// TIA Portal project "IMPERIAL" (V15)
// CUBE 67+ && PLC SIEMENS && ROBOT && PANTALLA GP-PRO

(* hardware
DEVICE "ROBOT1"  SIMATIC PC station
   slot 0: "Estación PC"  Rail  SIMATIC PC-Station  V1.0
      slot 125: "Stationmanager"  Station_Manager  V6.0.4
   slot 1: "CP 1616_1"  CP 1616  6GK1 161-6AA00  V2.6
DEVICE "Dispositivo GSD_1"  GSD.Device.PN
   slot 0: "Rack"  Rack  V1.0
   slot 0: "Cube67-BN-PNIO"  Cube67+ BN-PNIO  56526  2
      slot 0: "Cube67+ BN-PNIO_1"  Cube67+ BN-PNIO
      slot 1: "Cube67+ BN-PNIO"  Cube67+ BN-PNIO
         slot 1: "Puerto 1"  Port 1
         slot 2: "Puerto 2"  Port 2
      slot 1: "Alimentación de energía_1"  Power Supply
         slot 0: "Alimentación de energía"  Power Supply
   slot 3: "Rama 1_1"  Branch 0
      slot 0: "Rama 1"  Branch 0
   slot 4: "56601 DIO16 E 8xM12_1"  56601 DIO16 E 8xM12  56601
      slot 0: "56601 DIO16 E 8xM12"  56601 DIO16 E 8xM12
   slot 5: "Rama 2_1"  Branch 1
      slot 0: "Rama 2"  Branch 1
   slot 6: "56600 DIO16 C 8xM12_1"  56600 DIO16 C 8xM12  56600
      slot 0: "56600 DIO16 C 8xM12"  56600 DIO16 C 8xM12
   slot 7: "Rama 3_1"  Branch 2
      slot 0: "Rama 3"  Branch 2
   slot 8: "Rama 4_1"  Branch 3
      slot 0: "Rama 4"  Branch 3
DEVICE "S7-1200 station_1"  S7-1200 Station
   slot 0: "Rack_0"  S7-1200 Rack  Rack  V1.0
   slot 1: "PLC_1"  CPU 1212C DC/DC/DC  6ES7 212-1AE40-0XB0  V4.2
*)

// ===== PLC "PLC_1"  CPU 1212C DC/DC/DC =====

VAR_GLOBAL   // PLC tag table "Tabla de variables estándar"
   "PLC_C67_FOT_DAR_DARSENA2" AT %I29.7 : Bool;   // FOTO ESPEJO DAR 2
   "PLC_67_SME_DAR_DARSENA1" AT %I23.7 : Bool;   // FOTO DARSENA 1
   "R01_PLC_ORD_EXT_MDZ" AT %I10.0 : Bool;
   "R01_PLC_ORD_RET_MDZ" AT %I10.1 : Bool;
   "R01_PLC_PROD_COG_T1" AT %I10.2 : Bool;
   "NºSACOS" AT %IW30 : Word;
   "Nº DEJADAS CAPA PAR" AT %IW32 : Word;
   "Nº DEJADA CAPA IMPAR" AT %IW34 : Word;
   "ANCHO SACO" AT %IW36 : Word;
   "LARGO SACO" AT %IW38 : Word;
   "ALTO SACO" AT %IW40 : Word;
   "ANCHO PALET" AT %IW42 : Word;
   "LARGO PALET" AT %IW44 : Word;
   "ALTO PALET" AT %IW46 : Word;
   "X" AT %IW48 : Word;
   "Y" AT %IW50 : Word;
   "GIRO" AT %IB51 : Byte;
   "COGIDA" AT %I52.0 : Bool;
   "X(1)" AT %IW130 : Word;
   "Y(1)" AT %IW132 : Word;
   "GIRO(1)" AT %IB134 : Byte;
   "COGIDA(1)" AT %I135.0 : Bool;
   "X(2)" AT %IW136 : Word;
   "Y(2)" AT %IW138 : Word;
   "GIRO(2)" AT %IB140 : Byte;
   "COGIDA(2)" AT %I141.0 : Bool;
   "X(3)" AT %IW142 : Word;
   "Y(3)" AT %IW144 : Word;
   "GIRO(3)" AT %IB146 : Byte;
   "COGIDA(3)" AT %I147.0 : Bool;
   "X(4)" AT %IW148 : Word;
   "Y(4)" AT %IW150 : Word;
   "GIRO(4)" AT %IB152 : Byte;
   "COGIDA(4)" AT %I153.0 : Bool;
   "X(5)" AT %IW154 : Word;
   "Y(5)" AT %IW156 : Word;
   "GIRO(5)" AT %IB158 : Byte;
   "COGIDA(5)" AT %I159.0 : Bool;
   "X(6)" AT %IW160 : Word;
   "Y(6)" AT %IW162 : Word;
   "GIRO(6)" AT %IB164 : Byte;
   "COGIDA(6)" AT %I165.0 : Bool;
   "X(7)" AT %IW166 : Word;
   "Y(7)" AT %IW168 : Word;
   "GIRO(7)" AT %IB170 : Byte;
   "COGIDA(7)" AT %I171.0 : Bool;
   "X(10)" AT %IW172 : Word;
   "Y(10)" AT %IW174 : Word;
   "GIRO(10)" AT %IB176 : Byte;
   "COGIDA(10)" AT %I177.0 : Bool;
   "X(11)" AT %IW178 : Word;
   "Y(11)" AT %IW180 : Word;
   "GIRO(11)" AT %IB182 : Byte;
   "COGIDA(11)" AT %I183.0 : Bool;
   "X(12)" AT %IW184 : Word;
   "Y(12)" AT %IW186 : Word;
   "GIRO(12)" AT %IB188 : Byte;
   "COGIDA(12)" AT %I189.0 : Bool;
   "X(13)" AT %IW190 : Word;
   "Y(13)" AT %IW192 : Word;
   "GIRO(13)" AT %IB194 : Byte;
   "COGIDA(13)" AT %I195.0 : Bool;
   "X(14)" AT %IW196 : Word;
   "Y(14)" AT %IW198 : Word;
   "GIRO(14)" AT %IB200 : Byte;
   "COGIDA(14)" AT %I201.0 : Bool;
   "X(15)" AT %IW202 : Word;
   "Y(15)" AT %IW204 : Word;
   "GIRO(15)" AT %IB206 : Byte;
   "COGIDA(15)" AT %I207.0 : Bool;
   "X(16)" AT %IW208 : Word;
   "Y(16)" AT %IW210 : Word;
   "GIRO(16)" AT %IB212 : Byte;
   "COGIDA(16)" AT %I213.0 : Bool;
   "X(17)" AT %IW214 : Word;
   "Y(17)" AT %IW216 : Word;
   "GIRO(17)" AT %IB218 : Byte;
   "COGIDA(17)" AT %I219.0 : Bool;
   "TE_TRANSPORT_1" AT %I220.0 : Bool;
   "TE_TRANSPORT_2" AT %I220.1 : Bool;
   "Programa_Activo" AT %I11.1 : Bool;
   "Seguridades_R01_OK" AT %I11.0 : Bool;
   "Botonera_Boton_Rojo" AT %I0.0 : Bool;
   "Botonera_Boton_Verde" AT %I0.1 : Bool;
   "Botonera_Boton_Amarillo" AT %I0.2 : Bool;
   "R01_PLC_PROD_COG_T2" AT %I10.3 : Bool;
   "R01_PLC_ORD_EXT_PIS" AT %I10.4 : Bool;
   "R01_PLC_ROB_COG_T1" AT %I10.5 : Bool;
   "R01_PLC_ROB_COG_T2" AT %I10.6 : Bool;
   "R01_PLC_ORDEN_ABRIR" AT %Q19.1 : Bool;
   "R01_PLC_ORDEN_CERRAR" AT %Q19.2 : Bool;
   "P_On" AT %Q29.3 : Bool;
   "RESET_FLANCO_SUB" AT %Q29.5 : Bool;
   "PLC_R01_PERM_COG_SACO_T1" AT %Q10.2 : Bool;
   "PLC_R01_PERM_COG_SACO_T2" AT %Q10.3 : Bool;
   "Botonera_Luz_Roja" AT %Q0.0 : Bool;
   "Botonera_Luz_Verde" AT %Q0.1 : Bool;
   "Botonera_Luz_Amarillo" AT %Q0.2 : Bool;
   "R01_Boton_Rojo" AT %Q12.0 : Bool;
   "R01_Boton_Verde" AT %Q12.1 : Bool;
   "R01_Boton_Amarilla" AT %Q12.2 : Bool;
   "PLC_R01_PIS_EXT" AT %Q10.4 : Bool;
   "Orden_Abrir_Mordaza" AT %M200.0 : Bool;
   "Orden_Cerrar_Mordaza" AT %M200.1 : Bool;
   "Tag_8" AT %M200.3 : Bool;
   "Tag_8(1)" AT %M201.4 : Bool;
   "Tag_9" AT %M201.6 : Bool;
   "Tag_12(1)" AT %M201.7 : Bool;
   "Tag_10" AT %M202.0 : Bool;
   "Tag_13" AT %M202.1 : Bool;
   "Tag_11" AT %M202.2 : Bool;
   "Tag_100" AT %M202.3 : Bool;
   "LUZ_AMARILLA" AT %M202.4 : Bool;
   "LUZ_ROJA" AT %M202.5 : Bool;
   "LUZ_VERDE" AT %M202.6 : Bool;
   "Permiso_Meter_Saco" AT %M202.7 : Bool;
   "ERROR_GLOBAL" AT %M203.0 : Bool;
   "Seguridades_Armadas" AT %M201.0 : Bool;
   "PLC_C67_MDZ_RET_GAR" AT %Q21.6 : Bool;
   "PLC_C67_MDZ_EXT_GAR" AT %Q21.4 : Bool;
   "PLC_C67_EXT_P1" AT %Q21.2 : Bool;
   "PLC_C67_EXT_P2" AT %Q21.0 : Bool;
   "C67_PLC_SME_P2_RET" AT %I20.3 : Bool;
   "C67_PLC_SME_P2_EXT" AT %I21.3 : Bool;
   "C67_PLC_SME_P1_RET" AT %I20.1 : Bool;
   "C67_PLC_SME_P1_EXT" AT %I21.1 : Bool;
   "C67_PLC_SME_GARR_RET" AT %I21.5 : Bool;
   "C67_PLC_SME_GARR_EXT" AT %I20.5 : Bool;
   "PLC_C67_EXT_COST" AT %Q22.2 : Bool;
   "PLC_C67_MOT1_AVAN" AT %Q22.0 : Bool;
   "PLC_C67_MOT1_RET" AT %Q23.0 : Bool;
   "C67_PLC_FOTO_INICIO" AT %I23.3 : Bool;
   "C67_PLC_FOTO_FIN" AT %I23.1 : Bool;
   "C67_PLC_SME_COST_EXT" AT %I23.5 : Bool;
   "C67_PLC_SME_COST_RET" AT %I22.5 : Bool;
   "Tag_1" AT %I11.5 : Bool;
   "Tag_2" AT %Q11.4 : Bool;
   "Tag_3" AT %Q11.2 : Bool;
   "PLC_R01_MDZ_EXT" AT %Q10.0 : Bool;
   "PLC_R01_MDZ_RET" AT %Q10.1 : Bool;
END_VAR

DATA_BLOCK "DB_1"   // DB1
{ S7_Optimized_Access := 'FALSE' }
VERSION : 0.1
   VAR
      GP_SysStartAddress : Int;
   END_VAR
BEGIN
END_DATA_BLOCK

DATA_BLOCK "PISTON_EV_DB_1"   // DB2
{ S7_Optimized_Access := 'TRUE' }
VERSION : 0.1
// stored: InstanceOfName PISTON_EV
"PISTON_EV"
BEGIN
END_DATA_BLOCK

DATA_BLOCK "FUNCION_COGER_R01_DB_1"   // DB3
{ S7_Optimized_Access := 'TRUE' }
VERSION : 0.1
// stored: InstanceOfName FUNCION_COGER_R01
"FUNCION_COGER_R01"
BEGIN
END_DATA_BLOCK

DATA_BLOCK "FUNCION_PISADOR_DB"   // DB4
{ S7_Optimized_Access := 'TRUE' }
VERSION : 0.1
// stored: InstanceOfName FUNCION_PISADOR
"FUNCION_PISADOR"
BEGIN
END_DATA_BLOCK

DATA_BLOCK "FUNCION_COGER_R01_DB"   // DB5
{ S7_Optimized_Access := 'TRUE' }
VERSION : 0.1
// stored: InstanceOfName FUNCION_COGER_R01
"FUNCION_COGER_R01"
BEGIN
END_DATA_BLOCK

DATA_BLOCK "FUNCION_EV_DB"   // DB6
{ S7_Optimized_Access := 'TRUE' }
VERSION : 0.1
// stored: InstanceOfName FUNCION_EV
"FUNCION_EV"
BEGIN
END_DATA_BLOCK

DATA_BLOCK "FUNCION_EV_DB_1"   // DB7
{ S7_Optimized_Access := 'TRUE' }
VERSION : 0.1
// stored: InstanceOfName FUNCION_EV
"FUNCION_EV"
BEGIN
END_DATA_BLOCK

DATA_BLOCK "FUNCION_PISADOR_DB_1"   // DB8
{ S7_Optimized_Access := 'TRUE' }
VERSION : 0.1
// stored: InstanceOfName FUNCION_PISADOR
"FUNCION_PISADOR"
BEGIN
END_DATA_BLOCK

DATA_BLOCK "FUNCION_PISADOR_1_DB"   // DB9
{ S7_Optimized_Access := 'TRUE' }
VERSION : 0.1
// stored: InstanceOfName FUNCION_PISADOR
"FUNCION_PISADOR"
BEGIN
END_DATA_BLOCK

DATA_BLOCK "FUNCION_PISADOR_2_DB"   // DB10
{ S7_Optimized_Access := 'TRUE' }
VERSION : 0.1
// stored: InstanceOfName FUNCION_PISADOR
"FUNCION_PISADOR"
BEGIN
END_DATA_BLOCK

DATA_BLOCK "PISTON_EV_DB_2"   // DB11
{ S7_Optimized_Access := 'TRUE' }
VERSION : 0.1
// stored: InstanceOfName PISTON_EV
"PISTON_EV"
BEGIN
END_DATA_BLOCK

DATA_BLOCK "PISTON_EV_DB_3"   // DB12
{ S7_Optimized_Access := 'TRUE' }
VERSION : 0.1
// stored: InstanceOfName PISTON_EV
"PISTON_EV"
BEGIN
END_DATA_BLOCK

DATA_BLOCK "FUNCION_COGER_R01_DB_2"   // DB13
{ S7_Optimized_Access := 'TRUE' }
VERSION : 0.1
// stored: InstanceOfName FUNCION_COGER_R01
"FUNCION_COGER_R01"
BEGIN
END_DATA_BLOCK

DATA_BLOCK "FUNCION_COGER_R01_DB_3"   // DB14
{ S7_Optimized_Access := 'TRUE' }
VERSION : 0.1
// stored: InstanceOfName FUNCION_COGER_R01
"FUNCION_COGER_R01"
BEGIN
END_DATA_BLOCK

DATA_BLOCK "FUNCION_COGER_R01_DB_4"   // DB15
{ S7_Optimized_Access := 'TRUE' }
VERSION : 0.1
// stored: InstanceOfName FUNCION_COGER_R01
"FUNCION_COGER_R01"
BEGIN
END_DATA_BLOCK

DATA_BLOCK "FUNCION_COGER_R01_DB_5"   // DB16
{ S7_Optimized_Access := 'TRUE' }
VERSION : 0.1
// stored: InstanceOfName FUNCION_COGER_R01
"FUNCION_COGER_R01"
BEGIN
END_DATA_BLOCK

DATA_BLOCK "FUNCION_EV_DB_2"   // DB17
{ S7_Optimized_Access := 'TRUE' }
VERSION : 0.1
// stored: InstanceOfName FUNCION_EV
"FUNCION_EV"
BEGIN
END_DATA_BLOCK

DATA_BLOCK "FUNCION_PISADOR_DB_2"   // DB18
{ S7_Optimized_Access := 'TRUE' }
VERSION : 0.1
// stored: InstanceOfName FUNCION_PISADOR
"FUNCION_PISADOR"
BEGIN
END_DATA_BLOCK

DATA_BLOCK "FUNCION_PISADOR_DB_3"   // DB19
{ S7_Optimized_Access := 'TRUE' }
VERSION : 0.1
// stored: InstanceOfName FUNCION_PISADOR
"FUNCION_PISADOR"
BEGIN
END_DATA_BLOCK

DATA_BLOCK "FUNCION_EV_DB_3"   // DB20
{ S7_Optimized_Access := 'TRUE' }
VERSION : 0.1
// stored: InstanceOfName FUNCION_EV
"FUNCION_EV"
BEGIN
END_DATA_BLOCK

DATA_BLOCK "FUNCION_COGER_R01_DB_6"   // DB21
{ S7_Optimized_Access := 'TRUE' }
VERSION : 0.1
// stored: InstanceOfName FUNCION_COGER_R01
"FUNCION_COGER_R01"
BEGIN
END_DATA_BLOCK

DATA_BLOCK "PISTON_EV_DB"   // DB23
{ S7_Optimized_Access := 'TRUE' }
VERSION : 0.1
// stored: InstanceOfName PISTON_EV
"PISTON_EV"
BEGIN
END_DATA_BLOCK

DATA_BLOCK "TRANSPORTADOR_AUTOMATICO_DB"   // DB24
{ S7_Optimized_Access := 'TRUE' }
VERSION : 0.1
// stored: InstanceOfName TRANSPORTADOR_AUTOMATICO
"TRANSPORTADOR_AUTOMATICO"
BEGIN
END_DATA_BLOCK

DATA_BLOCK "FUNCION_EV_DB_8"   // DB25
{ S7_Optimized_Access := 'TRUE' }
VERSION : 0.1
// stored: InstanceOfName FUNCION_EV
"FUNCION_EV"
BEGIN
END_DATA_BLOCK

DATA_BLOCK "FUNCION_EV_DB_9"   // DB26
{ S7_Optimized_Access := 'TRUE' }
VERSION : 0.1
// stored: InstanceOfName FUNCION_EV
"FUNCION_EV"
BEGIN
END_DATA_BLOCK

DATA_BLOCK "FUNCION_EV_DB_4"   // DB30
{ S7_Optimized_Access := 'TRUE' }
VERSION : 0.1
// stored: InstanceOfName FUNCION_EV
"FUNCION_EV"
BEGIN
END_DATA_BLOCK

DATA_BLOCK "FUNCION_EV_DB_5"   // DB31
{ S7_Optimized_Access := 'TRUE' }
VERSION : 0.1
// stored: InstanceOfName FUNCION_EV
"FUNCION_EV"
BEGIN
END_DATA_BLOCK

DATA_BLOCK "PISTON_EV_DB_4"   // DB32
{ S7_Optimized_Access := 'TRUE' }
VERSION : 0.1
// stored: InstanceOfName PISTON_EV
"PISTON_EV"
BEGIN
END_DATA_BLOCK

DATA_BLOCK "PISTON_EV_DB_5"   // DB33
{ S7_Optimized_Access := 'TRUE' }
VERSION : 0.1
// stored: InstanceOfName PISTON_EV
"PISTON_EV"
BEGIN
END_DATA_BLOCK

DATA_BLOCK "FUNCION_EV_DB_6"   // DB34
{ S7_Optimized_Access := 'TRUE' }
VERSION : 0.1
// stored: InstanceOfName FUNCION_EV
"FUNCION_EV"
BEGIN
END_DATA_BLOCK

DATA_BLOCK "FUNCION_EV_DB_7"   // DB35
{ S7_Optimized_Access := 'TRUE' }
VERSION : 0.1
// stored: InstanceOfName FUNCION_EV
"FUNCION_EV"
BEGIN
END_DATA_BLOCK

DATA_BLOCK "EMPUJADOR_DB"   // DB36
{ S7_Optimized_Access := 'TRUE' }
VERSION : 0.1
// stored: InstanceOfName EMPUJADOR
"EMPUJADOR"
BEGIN
END_DATA_BLOCK

DATA_BLOCK "TRANSPORTADOR_AUTOMATICO_DB_1"   // DB37
{ S7_Optimized_Access := 'TRUE' }
VERSION : 0.1
// stored: InstanceOfName TRANSPORTADOR_AUTOMATICO
"TRANSPORTADOR_AUTOMATICO"
BEGIN
END_DATA_BLOCK

DATA_BLOCK "TRANSPORTADOR_AUTOMATICO_DB_2"   // DB38
{ S7_Optimized_Access := 'TRUE' }
VERSION : 0.1
// stored: InstanceOfName TRANSPORTADOR_AUTOMATICO
"TRANSPORTADOR_AUTOMATICO"
BEGIN
END_DATA_BLOCK

DATA_BLOCK "TRANSPORTADOR_AUTOMATICO_DB_3"   // DB39
{ S7_Optimized_Access := 'TRUE' }
VERSION : 0.1
// stored: InstanceOfName TRANSPORTADOR_AUTOMATICO
"TRANSPORTADOR_AUTOMATICO"
BEGIN
END_DATA_BLOCK

DATA_BLOCK "TRANSPORTADOR_AUTOMATICO_DB_4"   // DB40
{ S7_Optimized_Access := 'TRUE' }
VERSION : 0.1
// stored: InstanceOfName TRANSPORTADOR_AUTOMATICO
"TRANSPORTADOR_AUTOMATICO"
BEGIN
END_DATA_BLOCK

DATA_BLOCK "TRANSPORTADOR_AUTOMATICO_DB_5"   // DB41
{ S7_Optimized_Access := 'TRUE' }
VERSION : 0.1
// stored: InstanceOfName TRANSPORTADOR_AUTOMATICO
"TRANSPORTADOR_AUTOMATICO"
BEGIN
END_DATA_BLOCK

DATA_BLOCK "TRANSPORTADOR_AUTOMATICO_DB_6"   // DB42
{ S7_Optimized_Access := 'TRUE' }
VERSION : 0.1
// stored: InstanceOfName TRANSPORTADOR_AUTOMATICO
"TRANSPORTADOR_AUTOMATICO"
BEGIN
END_DATA_BLOCK

FUNCTION_BLOCK "PISTON_EV"   // FB1, LAD
TITLE = EV
{ S7_Optimized_Access := 'TRUE' }
VERSION : 0.1
   VAR_INPUT
      ORDEN_EXTENDER : Bool;
      ORDEN_RETRAER : Bool;
      SENSOR_EXTENDIDO : Bool;
      SENSOR_RETRAIDO : Bool;
   END_VAR
   VAR_OUTPUT
      CILINDRO_EXTENDIDO : Bool;
      EXTENDER_CILINDRO : Bool;
      CILINDRO_RETRAIDO : Bool;
      RETRAER_CILINDRO : Bool;
   END_VAR
BEGIN

REGION Network 1
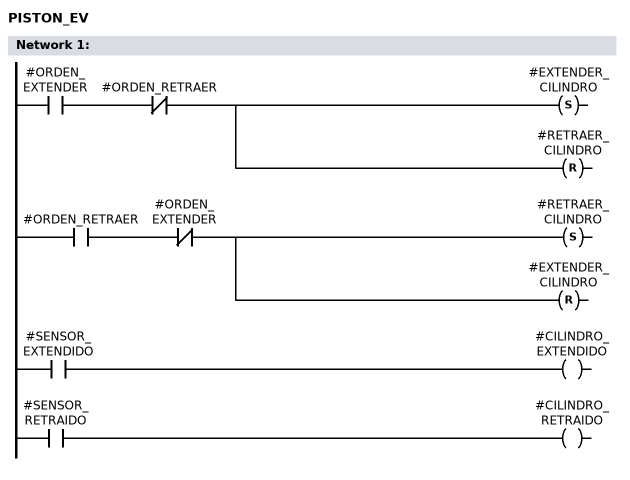
   RUNG wire#powerrail
      Contact( #ORDEN_EXTENDER )
      I_Contact( #ORDEN_RETRAER )
      wire#w1
      S_Coil( #EXTENDER_CILINDRO )
   END_RUNG
   RUNG wire#w1
      R_Coil( #RETRAER_CILINDRO )
   END_RUNG
   RUNG wire#powerrail
      Contact( #ORDEN_RETRAER )
      I_Contact( #ORDEN_EXTENDER )
      wire#w2
      S_Coil( #RETRAER_CILINDRO )
   END_RUNG
   RUNG wire#w2
      R_Coil( #EXTENDER_CILINDRO )
   END_RUNG
   RUNG wire#powerrail
      Contact( #SENSOR_EXTENDIDO )
      Coil( #CILINDRO_EXTENDIDO )
   END_RUNG
   RUNG wire#powerrail
      Contact( #SENSOR_RETRAIDO )
      Coil( #CILINDRO_RETRAIDO )
   END_RUNG
   // the same network as SCL:
   IF #ORDEN_EXTENDER AND NOT #ORDEN_RETRAER THEN
       #EXTENDER_CILINDRO := TRUE;
       #RETRAER_CILINDRO := FALSE;
   END_IF;
   IF #ORDEN_RETRAER AND NOT #ORDEN_EXTENDER THEN
       #RETRAER_CILINDRO := TRUE;
       #EXTENDER_CILINDRO := FALSE;
   END_IF;
   #CILINDRO_EXTENDIDO := #SENSOR_EXTENDIDO;
   #CILINDRO_RETRAIDO := #SENSOR_RETRAIDO;
END_REGION
END_FUNCTION_BLOCK

FUNCTION_BLOCK "FUNCION_EV"   // FB2, LAD
{ S7_Optimized_Access := 'TRUE' }
VERSION : 0.1
   VAR_INPUT
      Orden_Retraer_Pistones : Bool;   // INPUT
      Orden_Extender_Pistones : Bool;   // INPUT
      Sensor_1_Extendido : Bool;   // INPUT
      Sensor_1_Retraido : Bool;   // INPUT
      Sensor_2_Extendido : Bool;   // INPUT
      Sensor_2_Retraido : Bool;   // INPUT
      EN_Piston_Doble : Bool;   // INPUT
      EN_Switch_Final_Carrera_Retraer : Bool;   // INPUT
      EN_Switch_Final_Carrera_Extender : Bool;   // INPUT
      Tiempo_Error_Extender_100ms : Time := T#100ms;   // 0
      Tiempo_Error_Retraer_100ms : Time := T#100ms;   // 0
   END_VAR
   VAR_OUTPUT
      Error_Extender : Bool;   // OUTPUT
      Error_Retroceder : Bool;   // OUTPUT
      Extender_Pistones : Bool;
      Retraer_Pistones : Bool;
      Pistones_Retraidos : Bool;
      Pistones_Extendidos : Bool;
   END_VAR
   VAR
      Extender_Piston_1 : Bool;   // INTERNAL
      Extender_Piston_2 : Bool;   // INTERNAL
      Retraer_Piston_1 : Bool;   // INTERNAL
      Retraer_Piston_2 : Bool;   // INTERNAL
      Piston_1_Extendido : Bool;   // INTERNAL
      Piston_1_Retraido : Bool;   // INTERNAL
      Piston_2_Extendido : Bool;   // INTERNAL
      Piston_2_Retraido : Bool;   // INTERNAL
      Piston_1 : "PISTON_EV";
      Piston_2 : "PISTON_EV";
      Timer_1 : Time;   // INTERNAL
      Timer_2 : Time;   // INTERNAL
   END_VAR
BEGIN

REGION Network 1
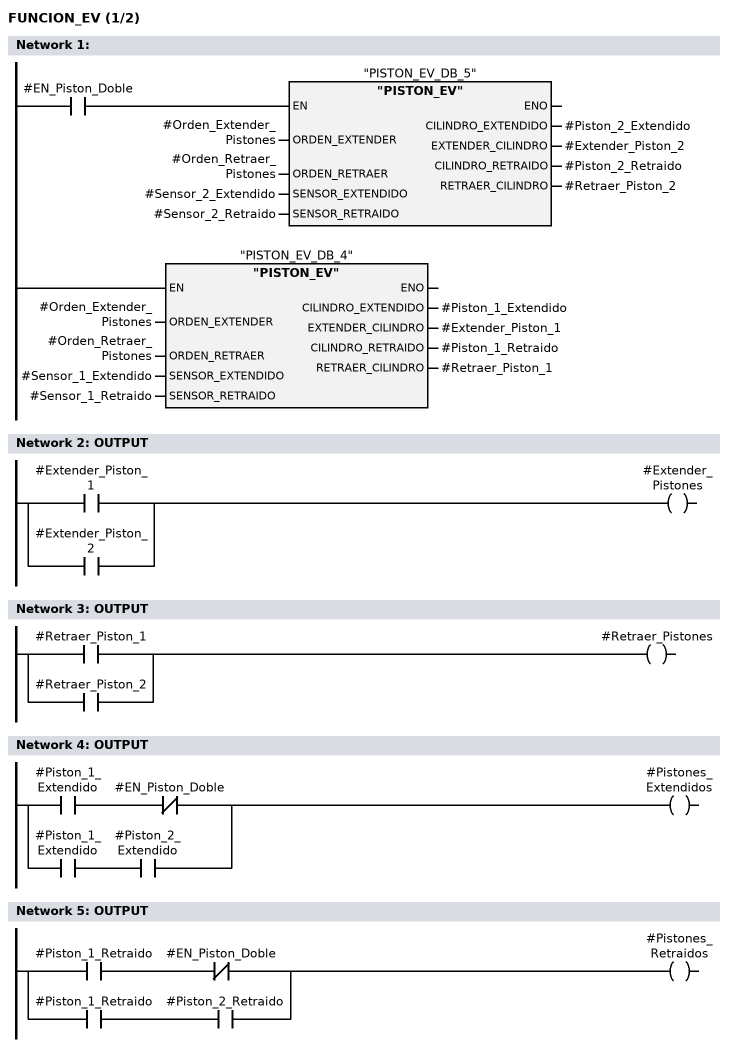
   RUNG wire#powerrail
      Contact( #EN_Piston_Doble )
      "PISTON_EV_DB_5"(ORDEN_EXTENDER := #Orden_Extender_Pistones, ORDEN_RETRAER := #Orden_Retraer_Pistones, SENSOR_EXTENDIDO := #Sensor_2_Extendido, SENSOR_RETRAIDO := #Sensor_2_Retraido, CILINDRO_EXTENDIDO => #Piston_2_Extendido, EXTENDER_CILINDRO => #Extender_Piston_2, CILINDRO_RETRAIDO => #Piston_2_Retraido, RETRAER_CILINDRO => #Retraer_Piston_2)
   END_RUNG
   RUNG wire#powerrail
      "PISTON_EV_DB_4"(ORDEN_EXTENDER := #Orden_Extender_Pistones, ORDEN_RETRAER := #Orden_Retraer_Pistones, SENSOR_EXTENDIDO := #Sensor_1_Extendido, SENSOR_RETRAIDO := #Sensor_1_Retraido, CILINDRO_EXTENDIDO => #Piston_1_Extendido, EXTENDER_CILINDRO => #Extender_Piston_1, CILINDRO_RETRAIDO => #Piston_1_Retraido, RETRAER_CILINDRO => #Retraer_Piston_1)
   END_RUNG
   // the same network as SCL:
   IF #EN_Piston_Doble THEN
       "PISTON_EV_DB_5"(ORDEN_EXTENDER := #Orden_Extender_Pistones,   // "PISTON_EV"
                        ORDEN_RETRAER := #Orden_Retraer_Pistones,
                        SENSOR_EXTENDIDO := #Sensor_2_Extendido,
                        SENSOR_RETRAIDO := #Sensor_2_Retraido,
                        CILINDRO_EXTENDIDO => #Piston_2_Extendido,
                        EXTENDER_CILINDRO => #Extender_Piston_2,
                        CILINDRO_RETRAIDO => #Piston_2_Retraido,
                        RETRAER_CILINDRO => #Retraer_Piston_2);
   END_IF;
   "PISTON_EV_DB_4"(ORDEN_EXTENDER := #Orden_Extender_Pistones,   // "PISTON_EV"
                    ORDEN_RETRAER := #Orden_Retraer_Pistones,
                    SENSOR_EXTENDIDO := #Sensor_1_Extendido,
                    SENSOR_RETRAIDO := #Sensor_1_Retraido,
                    CILINDRO_EXTENDIDO => #Piston_1_Extendido,
                    EXTENDER_CILINDRO => #Extender_Piston_1,
                    CILINDRO_RETRAIDO => #Piston_1_Retraido,
                    RETRAER_CILINDRO => #Retraer_Piston_1);
END_REGION

REGION Network 2: OUTPUT
   RUNG wire#powerrail
      Contact( #Extender_Piston_1 )
      wire#w1
      Coil( #Extender_Pistones )
   END_RUNG
   RUNG wire#powerrail
      Contact( #Extender_Piston_2 )
   END_RUNG wire#w1
   // the same network as SCL:
   #Extender_Pistones := #Extender_Piston_1 OR #Extender_Piston_2;
END_REGION

REGION Network 3: OUTPUT
   RUNG wire#powerrail
      Contact( #Retraer_Piston_1 )
      wire#w1
      Coil( #Retraer_Pistones )
   END_RUNG
   RUNG wire#powerrail
      Contact( #Retraer_Piston_2 )
   END_RUNG wire#w1
   // the same network as SCL:
   #Retraer_Pistones := #Retraer_Piston_1 OR #Retraer_Piston_2;
END_REGION

REGION Network 4: OUTPUT
   RUNG wire#powerrail
      Contact( #Piston_1_Extendido )
      I_Contact( #EN_Piston_Doble )
      wire#w1
      Coil( #Pistones_Extendidos )
   END_RUNG
   RUNG wire#powerrail
      Contact( #Piston_1_Extendido )
      Contact( #Piston_2_Extendido )
   END_RUNG wire#w1
   // the same network as SCL:
   #Pistones_Extendidos := (#Piston_1_Extendido AND NOT #EN_Piston_Doble) OR (#Piston_1_Extendido AND #Piston_2_Extendido);
END_REGION

REGION Network 5: OUTPUT
   RUNG wire#powerrail
      Contact( #Piston_1_Retraido )
      I_Contact( #EN_Piston_Doble )
      wire#w1
      Coil( #Pistones_Retraidos )
   END_RUNG
   RUNG wire#powerrail
      Contact( #Piston_1_Retraido )
      Contact( #Piston_2_Retraido )
   END_RUNG wire#w1
   // the same network as SCL:
   #Pistones_Retraidos := (#Piston_1_Retraido AND NOT #EN_Piston_Doble) OR (#Piston_1_Retraido AND #Piston_2_Retraido);
END_REGION

REGION Network 6: ERRORES 1: Si tarda más de 1s entre que doy la orden de extender y uno/dos de los cilindros no llegan al final de carrera, ó si la variable EN_Variable_Error esta on y uno/dos cilindros llegan al final de carrera.
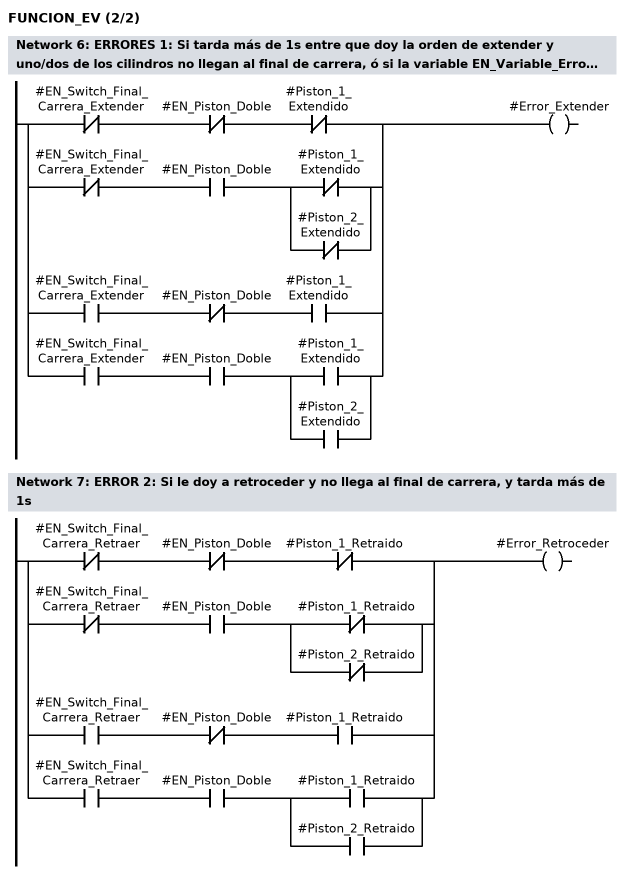
   RUNG wire#powerrail
      I_Contact( #EN_Switch_Final_Carrera_Extender )
      I_Contact( #EN_Piston_Doble )
      I_Contact( #Piston_1_Extendido )
      wire#w1
      Coil( #Error_Extender )
   END_RUNG
   RUNG wire#powerrail
      I_Contact( #EN_Switch_Final_Carrera_Extender )
      Contact( #EN_Piston_Doble )
      wire#w2
      I_Contact( #Piston_1_Extendido )
   END_RUNG wire#w1
   RUNG wire#w2
      I_Contact( #Piston_2_Extendido )
   END_RUNG wire#w1
   RUNG wire#powerrail
      Contact( #EN_Switch_Final_Carrera_Extender )
      I_Contact( #EN_Piston_Doble )
      Contact( #Piston_1_Extendido )
   END_RUNG wire#w1
   RUNG wire#powerrail
      Contact( #EN_Switch_Final_Carrera_Extender )
      Contact( #EN_Piston_Doble )
      wire#w3
      Contact( #Piston_1_Extendido )
   END_RUNG wire#w1
   RUNG wire#w3
      Contact( #Piston_2_Extendido )
   END_RUNG wire#w1
   // the same network as SCL:
   #Error_Extender := (NOT #EN_Switch_Final_Carrera_Extender AND NOT #EN_Piston_Doble AND NOT #Piston_1_Extendido) OR (NOT #EN_Switch_Final_Carrera_Extender AND #EN_Piston_Doble AND (NOT #Piston_1_Extendido OR NOT #Piston_2_Extendido)) OR (#EN_Switch_Final_Carrera_Extender AND NOT #EN_Piston_Doble AND #Piston_1_Extendido) OR (#EN_Switch_Final_Carrera_Extender AND #EN_Piston_Doble AND (#Piston_1_Extendido OR #Piston_2_Extendido));
END_REGION

REGION Network 7: ERROR 2: Si le doy a retroceder y no llega al final de carrera, y tarda más de 1s
   RUNG wire#powerrail
      I_Contact( #EN_Switch_Final_Carrera_Retraer )
      I_Contact( #EN_Piston_Doble )
      I_Contact( #Piston_1_Retraido )
      wire#w1
      Coil( #Error_Retroceder )
   END_RUNG
   RUNG wire#powerrail
      I_Contact( #EN_Switch_Final_Carrera_Retraer )
      Contact( #EN_Piston_Doble )
      wire#w2
      I_Contact( #Piston_1_Retraido )
   END_RUNG wire#w1
   RUNG wire#w2
      I_Contact( #Piston_2_Retraido )
   END_RUNG wire#w1
   RUNG wire#powerrail
      Contact( #EN_Switch_Final_Carrera_Retraer )
      I_Contact( #EN_Piston_Doble )
      Contact( #Piston_1_Retraido )
   END_RUNG wire#w1
   RUNG wire#powerrail
      Contact( #EN_Switch_Final_Carrera_Retraer )
      Contact( #EN_Piston_Doble )
      wire#w3
      Contact( #Piston_1_Retraido )
   END_RUNG wire#w1
   RUNG wire#w3
      Contact( #Piston_2_Retraido )
   END_RUNG wire#w1
   // the same network as SCL:
   #Error_Retroceder := (NOT #EN_Switch_Final_Carrera_Retraer AND NOT #EN_Piston_Doble AND NOT #Piston_1_Retraido) OR (NOT #EN_Switch_Final_Carrera_Retraer AND #EN_Piston_Doble AND (NOT #Piston_1_Retraido OR NOT #Piston_2_Retraido)) OR (#EN_Switch_Final_Carrera_Retraer AND NOT #EN_Piston_Doble AND #Piston_1_Retraido) OR (#EN_Switch_Final_Carrera_Retraer AND #EN_Piston_Doble AND (#Piston_1_Retraido OR #Piston_2_Retraido));
END_REGION
END_FUNCTION_BLOCK

FUNCTION_BLOCK "TRANSPORTADOR_AUTOMATICO"   // FB4, LAD
{ S7_Optimized_Access := 'TRUE' }
VERSION : 0.1
   VAR_INPUT
      Foto_Inicio : Bool;
      Foto_FIn : Bool;
      RESET : Bool;
      Producto_Cogido : Bool;
      Costillas_Subida : Bool;
      Costillas_Bajadas : Bool;
      Tiempo_Error_Saco_100ms : Time := T#100ms;
      Tiempo_Ahorro : Time := T#1000ms;
      Tiempo_Saco : Time := T#1000ms;
      Tiempo_No_Saco : Time := T#10000ms;
      Tiempo_Pegar_Saco : Time := T#200ms;
   END_VAR
   VAR_OUTPUT
      Orden_Extender_Costilla : Bool;
      Permiso_Meter_Saco : Bool;
      Permiso_Coger_Saco : Bool;
      Error_Saco : Bool;
      Motor : Bool;
   END_VAR
   VAR_IN_OUT
      Estado_Transportador : Int;
   END_VAR
   VAR
      IEC_Timer_0_DB_1 : TON_TIME;
      IEC_Timer_0_DB_2 : TON_TIME;
      IEC_Timer_0_DB_3 : TON_TIME;
      IEC_Timer_0_DB : TON_TIME;
      Timer1 : TON_TIME;
      Timer2 : TON_TIME;
      Timer3 : TON_TIME;
      Timer4 : TON_TIME;
      Timer5 : TON_TIME;
   END_VAR
BEGIN

REGION Network 1
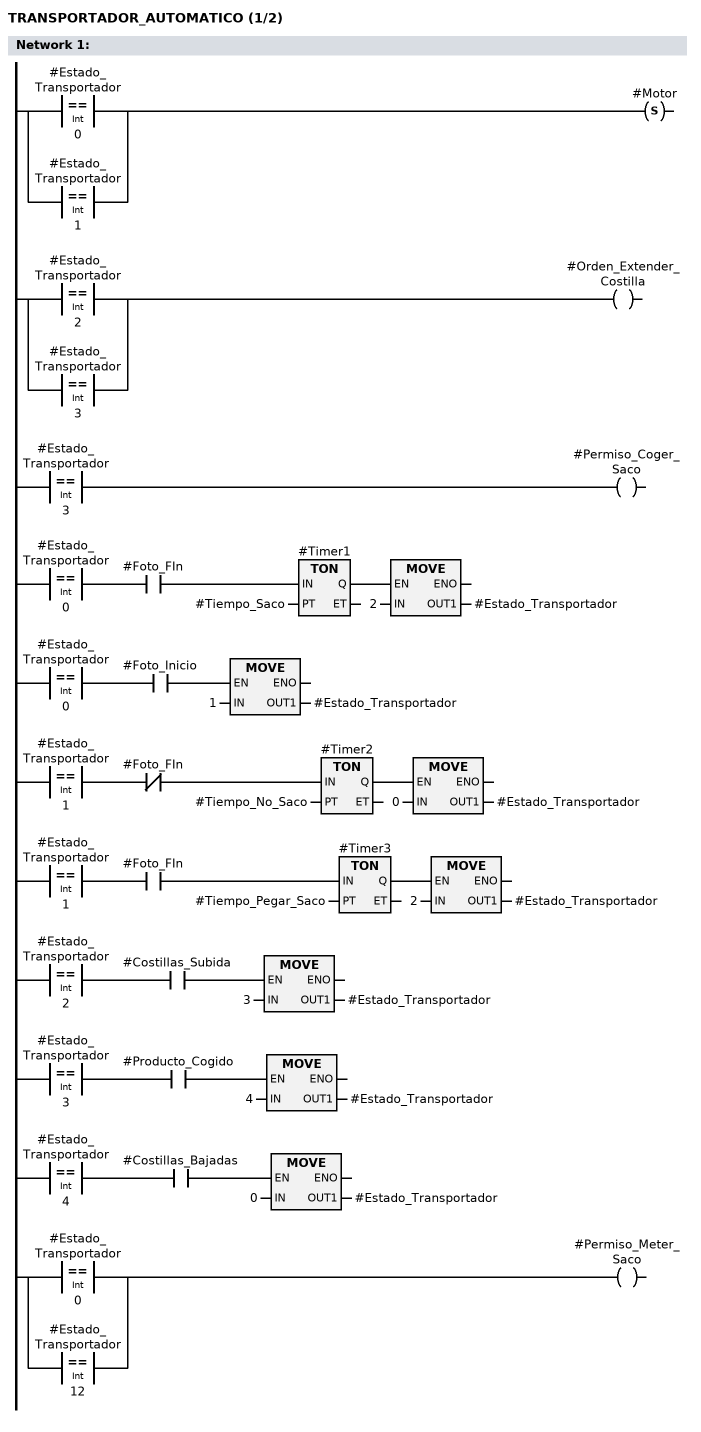
   IF (#Estado_Transportador = 0) OR (#Estado_Transportador = 1) THEN #Motor := TRUE; END_IF;
   #Orden_Extender_Costilla := (#Estado_Transportador = 2) OR (#Estado_Transportador = 3);
   #Permiso_Coger_Saco := #Estado_Transportador = 3;
   #Timer1(IN := (#Estado_Transportador = 0) AND #Foto_FIn, PT := #Tiempo_Saco);   // TON
   IF #Timer1.Q THEN #Estado_Transportador := 2; END_IF;
   IF (#Estado_Transportador = 0) AND #Foto_Inicio THEN #Estado_Transportador := 1; END_IF;
   #Timer2(IN := (#Estado_Transportador = 1) AND NOT #Foto_FIn, PT := #Tiempo_No_Saco);   // TON
   IF #Timer2.Q THEN #Estado_Transportador := 0; END_IF;
   #Timer3(IN := (#Estado_Transportador = 1) AND #Foto_FIn, PT := #Tiempo_Pegar_Saco);   // TON
   IF #Timer3.Q THEN #Estado_Transportador := 2; END_IF;
   IF (#Estado_Transportador = 2) AND #Costillas_Subida THEN #Estado_Transportador := 3; END_IF;
   IF (#Estado_Transportador = 3) AND #Producto_Cogido THEN #Estado_Transportador := 4; END_IF;
   IF (#Estado_Transportador = 4) AND #Costillas_Bajadas THEN #Estado_Transportador := 0; END_IF;
   #Permiso_Meter_Saco := (#Estado_Transportador = 0) OR (#Estado_Transportador = 12);
END_REGION

REGION Network 2
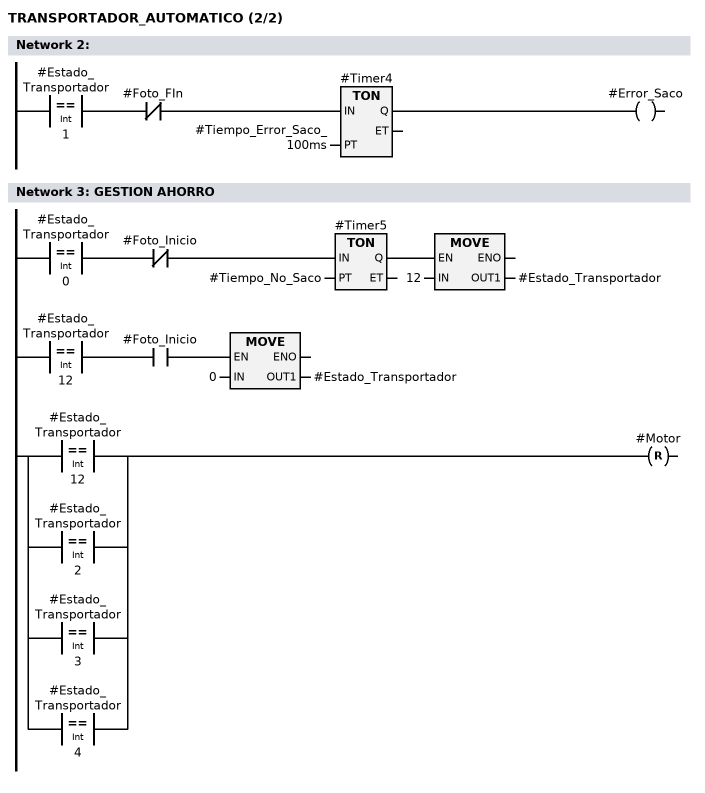
   #Timer4(IN := (#Estado_Transportador = 1) AND NOT #Foto_FIn, PT := #Tiempo_Error_Saco_100ms);   // TON
   #Error_Saco := #Timer4.Q;
END_REGION

REGION Network 3: GESTION AHORRO
   #Timer5(IN := (#Estado_Transportador = 0) AND NOT #Foto_Inicio, PT := #Tiempo_No_Saco);   // TON
   IF #Timer5.Q THEN #Estado_Transportador := 12; END_IF;
   IF (#Estado_Transportador = 12) AND #Foto_Inicio THEN #Estado_Transportador := 0; END_IF;
   IF (#Estado_Transportador = 12) OR (#Estado_Transportador = 2) OR (#Estado_Transportador = 3) OR (#Estado_Transportador = 4) THEN
       #Motor := FALSE;
   END_IF;
END_REGION
END_FUNCTION_BLOCK

FUNCTION_BLOCK "FUNCION_COGER_R01"   // FB5, LAD
{ S7_Optimized_Access := 'TRUE' }
VERSION : 0.1
   VAR_INPUT
      Orden_Cerrar_Garras : Bool;   // INPUT
      Orden_Abrir_Garras : Bool;   // INPUT
      SME_Garras_Cerradas : Bool;   // INPUT
      SME_garras_Abiertas : Bool;   // INPUT
      SME_Pisador_1_Abierto : Bool;
      SME_Pisador_1_Cerrado : Bool;
      SME_Pisador_2_Abierto : Bool;
      SME_Pisador_2_Cerrado : Bool;
      EN_1 : Bool;
   END_VAR
   VAR_OUTPUT
      Ok_Coger_1 : Bool;
      ENO_2 : Bool;
      Error_Coger_1 : Bool;
      Garras_Abierta_1 : Bool;
      Garras_Cerrada_1 : Bool;
      Pisador_1_Bajado : Bool;
      Pisador_2_Bajado : Bool;
      Pisador_1_Abierto : Bool;
      Pisador_2_Abierto : Bool;
   END_VAR
   VAR_IN_OUT
      Abrir_Garra_1 : Bool;
      Cerrar_Garra_1 : Bool;
      Abrir_Pisador_1 : Bool;
      Cerrar_Pisador_1 : Bool;
      Abrir_Pisador_2 : Bool;
      Cerrar_Pisador_2 : Bool;
   END_VAR
   VAR
      Orden_Abrir_Mordaza : Bool;
      Orden_Cerrar_Mordaza : Bool;
   END_VAR
BEGIN

REGION Network 1
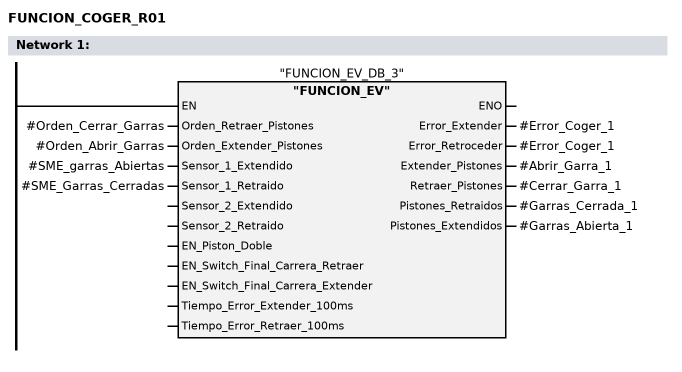
   RUNG wire#powerrail
      "FUNCION_EV_DB_3"(Orden_Retraer_Pistones := #Orden_Cerrar_Garras, Orden_Extender_Pistones := #Orden_Abrir_Garras, Sensor_1_Extendido := #SME_garras_Abiertas, Sensor_1_Retraido := #SME_Garras_Cerradas, Sensor_2_Extendido :=, Sensor_2_Retraido :=, EN_Piston_Doble :=, EN_Switch_Final_Carrera_Retraer :=, EN_Switch_Final_Carrera_Extender :=, Tiempo_Error_Extender_100ms :=, Tiempo_Error_Retraer_100ms :=, Error_Extender => #Error_Coger_1, Error_Retroceder => #Error_Coger_1, Extender_Pistones => #Abrir_Garra_1, Retraer_Pistones => #Cerrar_Garra_1, Pistones_Retraidos => #Garras_Cerrada_1, Pistones_Extendidos => #Garras_Abierta_1)
   END_RUNG
   // the same network as SCL:
   "FUNCION_EV_DB_3"(Orden_Retraer_Pistones := #Orden_Cerrar_Garras,   // "FUNCION_EV"
                     Orden_Extender_Pistones := #Orden_Abrir_Garras,
                     Sensor_1_Extendido := #SME_garras_Abiertas,
                     Sensor_1_Retraido := #SME_Garras_Cerradas,
                     Error_Extender => #Error_Coger_1,
                     Error_Retroceder => #Error_Coger_1,
                     Extender_Pistones => #Abrir_Garra_1,
                     Retraer_Pistones => #Cerrar_Garra_1,
                     Pistones_Retraidos => #Garras_Cerrada_1,
                     Pistones_Extendidos => #Garras_Abierta_1);
END_REGION
END_FUNCTION_BLOCK

FUNCTION_BLOCK "FUNCION_PISADOR"   // FB6, LAD
{ S7_Optimized_Access := 'TRUE' }
VERSION : 0.1
   VAR_INPUT
      Orden_Bajar_Pisador : Bool;
      Orden_Subir_Pisador : Bool;
      SME_Pisador_Bajado : Bool;
      SME_Pisador_Subido : Bool;
      EN_1 : Bool;
   END_VAR
   VAR_OUTPUT
      Ok_Coger_2 : Bool;
      ENO_1 : Bool;
      Error_Coger_2 : Bool;
   END_VAR
   VAR_IN_OUT
      Bajar_Pisador : Bool;
      Subir_Pisador : Bool;
   END_VAR
   VAR
      Pisador_Bajado_1 : Bool;
      Pisador_Subido_1 : Bool;
   END_VAR
BEGIN

REGION Network 1
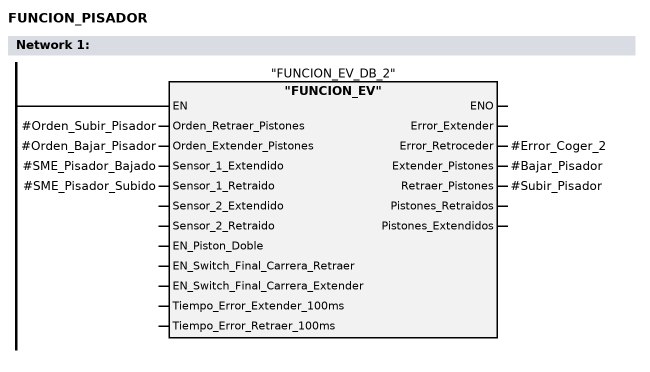
   RUNG wire#powerrail
      "FUNCION_EV_DB_2"(Orden_Retraer_Pistones := #Orden_Subir_Pisador, Orden_Extender_Pistones := #Orden_Bajar_Pisador, Sensor_1_Extendido := #SME_Pisador_Bajado, Sensor_1_Retraido := #SME_Pisador_Subido, Sensor_2_Extendido :=, Sensor_2_Retraido :=, EN_Piston_Doble :=, EN_Switch_Final_Carrera_Retraer :=, EN_Switch_Final_Carrera_Extender :=, Tiempo_Error_Extender_100ms :=, Tiempo_Error_Retraer_100ms :=, Extender_Pistones => #Bajar_Pisador, Retraer_Pistones => #Subir_Pisador, Error_Extender =>, Error_Retroceder => #Error_Coger_2, Pistones_Retraidos =>, Pistones_Extendidos =>)
   END_RUNG
   // the same network as SCL:
   "FUNCION_EV_DB_2"(Orden_Retraer_Pistones := #Orden_Subir_Pisador,   // "FUNCION_EV"
                     Orden_Extender_Pistones := #Orden_Bajar_Pisador,
                     Sensor_1_Extendido := #SME_Pisador_Bajado,
                     Sensor_1_Retraido := #SME_Pisador_Subido,
                     Error_Retroceder => #Error_Coger_2,
                     Extender_Pistones => #Bajar_Pisador,
                     Retraer_Pistones => #Subir_Pisador);
END_REGION
END_FUNCTION_BLOCK

FUNCTION_BLOCK "EMPUJADOR"   // FB7, LAD
{ S7_Optimized_Access := 'TRUE' }
VERSION : 0.1
   VAR_INPUT
      Foto_Inicio : Bool;
      SME_Empujar_Extendido : Bool;
      SME_Empujador_Retraido : Bool;
      Quiero_Saco_Empujador : Bool;
   END_VAR
   VAR_OUTPUT
      Extender_Empujador : Bool;
   END_VAR
   VAR_IN_OUT
      Estado_Transportador : Int;
      Retraer_Empujador : Bool;
   END_VAR
   VAR
      Orden_extender : Bool;
      Orden_retraer : Bool;
   END_VAR
BEGIN

REGION Network 1
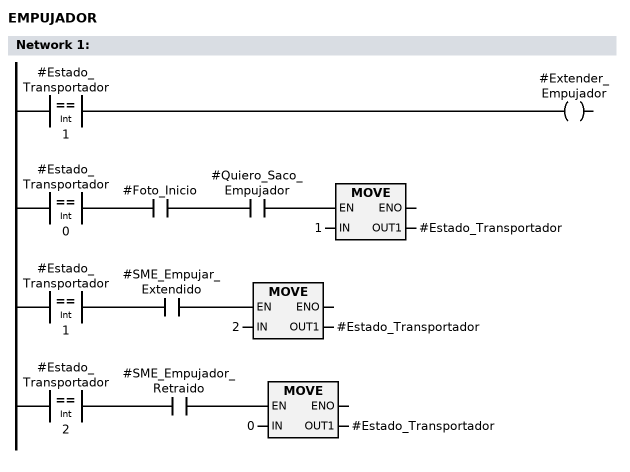
   RUNG wire#powerrail
      { S7_Templates := "SrcType := Int" } EQ_Contact(in1 := #Estado_Transportador, in2 := 1)
      Coil( #Extender_Empujador )
   END_RUNG
   RUNG wire#powerrail
      { S7_Templates := "SrcType := Int" } EQ_Contact(in1 := #Estado_Transportador, in2 := 0)
      Contact( #Foto_Inicio )
      Contact( #Quiero_Saco_Empujador )
      Move(in := 1, out1 => #Estado_Transportador)
   END_RUNG
   RUNG wire#powerrail
      { S7_Templates := "SrcType := Int" } EQ_Contact(in1 := #Estado_Transportador, in2 := 1)
      Contact( #SME_Empujar_Extendido )
      Move(in := 2, out1 => #Estado_Transportador)
   END_RUNG
   RUNG wire#powerrail
      { S7_Templates := "SrcType := Int" } EQ_Contact(in1 := #Estado_Transportador, in2 := 2)
      Contact( #SME_Empujador_Retraido )
      Move(in := 0, out1 => #Estado_Transportador)
   END_RUNG
   // the same network as SCL:
   #Extender_Empujador := #Estado_Transportador = 1;
   IF (#Estado_Transportador = 0) AND #Foto_Inicio AND #Quiero_Saco_Empujador THEN
       #Estado_Transportador := 1;
   END_IF;
   IF (#Estado_Transportador = 1) AND #SME_Empujar_Extendido THEN #Estado_Transportador := 2; END_IF;
   IF (#Estado_Transportador = 2) AND #SME_Empujador_Retraido THEN #Estado_Transportador := 0; END_IF;
END_REGION
END_FUNCTION_BLOCK

FUNCTION "BALIZA" : Void   // FC1, LAD
TITLE = BOTONERA
{ S7_Optimized_Access := 'TRUE' }
VERSION : 0.1
   VAR_INPUT
      Programa_Activo : Bool;
      Seguridades_Armadas : Bool;
      Seguridades_Robot_OK : Bool;
   END_VAR
BEGIN

REGION Network 1: LV
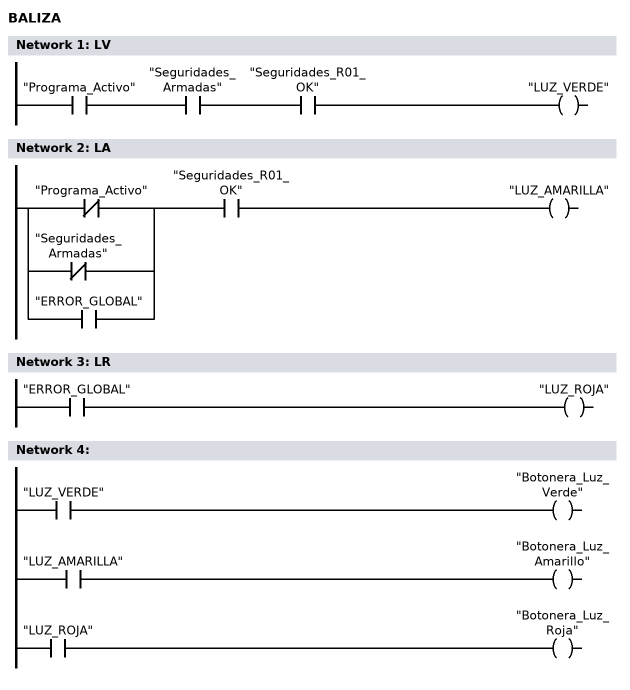
   RUNG wire#powerrail
      Contact( "Programa_Activo" )
      Contact( "Seguridades_Armadas" )
      Contact( "Seguridades_R01_OK" )
      Coil( "LUZ_VERDE" )
   END_RUNG
   // the same network as SCL:
   "LUZ_VERDE" := "Programa_Activo" AND "Seguridades_Armadas" AND "Seguridades_R01_OK";
END_REGION

REGION Network 2: LA
   RUNG wire#powerrail
      I_Contact( "Programa_Activo" )
      wire#w1
      Contact( "Seguridades_R01_OK" )
      Coil( "LUZ_AMARILLA" )
   END_RUNG
   RUNG wire#powerrail
      I_Contact( "Seguridades_Armadas" )
   END_RUNG wire#w1
   RUNG wire#powerrail
      Contact( "ERROR_GLOBAL" )
   END_RUNG wire#w1
   // the same network as SCL:
   "LUZ_AMARILLA" := (NOT "Programa_Activo" OR NOT "Seguridades_Armadas" OR "ERROR_GLOBAL") AND "Seguridades_R01_OK";
END_REGION

REGION Network 3: LR
   RUNG wire#powerrail
      Contact( "ERROR_GLOBAL" )
      Coil( "LUZ_ROJA" )
   END_RUNG
   // the same network as SCL:
   "LUZ_ROJA" := "ERROR_GLOBAL";
END_REGION

REGION Network 4
   RUNG wire#powerrail
      Contact( "LUZ_VERDE" )
      Coil( "Botonera_Luz_Verde" )
   END_RUNG
   RUNG wire#powerrail
      Contact( "LUZ_AMARILLA" )
      Coil( "Botonera_Luz_Amarillo" )
   END_RUNG
   RUNG wire#powerrail
      Contact( "LUZ_ROJA" )
      Coil( "Botonera_Luz_Roja" )
   END_RUNG
   // the same network as SCL:
   "Botonera_Luz_Verde" := "LUZ_VERDE";
   "Botonera_Luz_Amarillo" := "LUZ_AMARILLA";
   "Botonera_Luz_Roja" := "LUZ_ROJA";
END_REGION
END_FUNCTION

FUNCTION "BOTONERA" : Void   // FC2, LAD
{ S7_Optimized_Access := 'TRUE' }
VERSION : 0.1
BEGIN

REGION Network 1
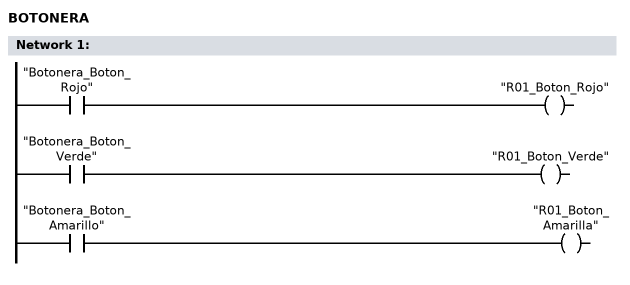
   RUNG wire#powerrail
      Contact( "Botonera_Boton_Rojo" )
      Coil( "R01_Boton_Rojo" )
   END_RUNG
   RUNG wire#powerrail
      Contact( "Botonera_Boton_Verde" )
      Coil( "R01_Boton_Verde" )
   END_RUNG
   RUNG wire#powerrail
      Contact( "Botonera_Boton_Amarillo" )
      Coil( "R01_Boton_Amarilla" )
   END_RUNG
   // the same network as SCL:
   "R01_Boton_Rojo" := "Botonera_Boton_Rojo";
   "R01_Boton_Verde" := "Botonera_Boton_Verde";
   "R01_Boton_Amarilla" := "Botonera_Boton_Amarillo";
END_REGION
END_FUNCTION

ORGANIZATION_BLOCK "Main"   // OB1, LAD, ProgramCycle
TITLE = "Main Program Sweep (Cycle)"
{ S7_Optimized_Access := 'TRUE' }
VERSION : 0.1
   VAR_INPUT
      Initial_Call : Bool;   // Initial call of this OB
      Remanence : Bool;   // =True, if remanent data are available
   END_VAR
BEGIN

REGION Network 1: MORDAZA ROBOT
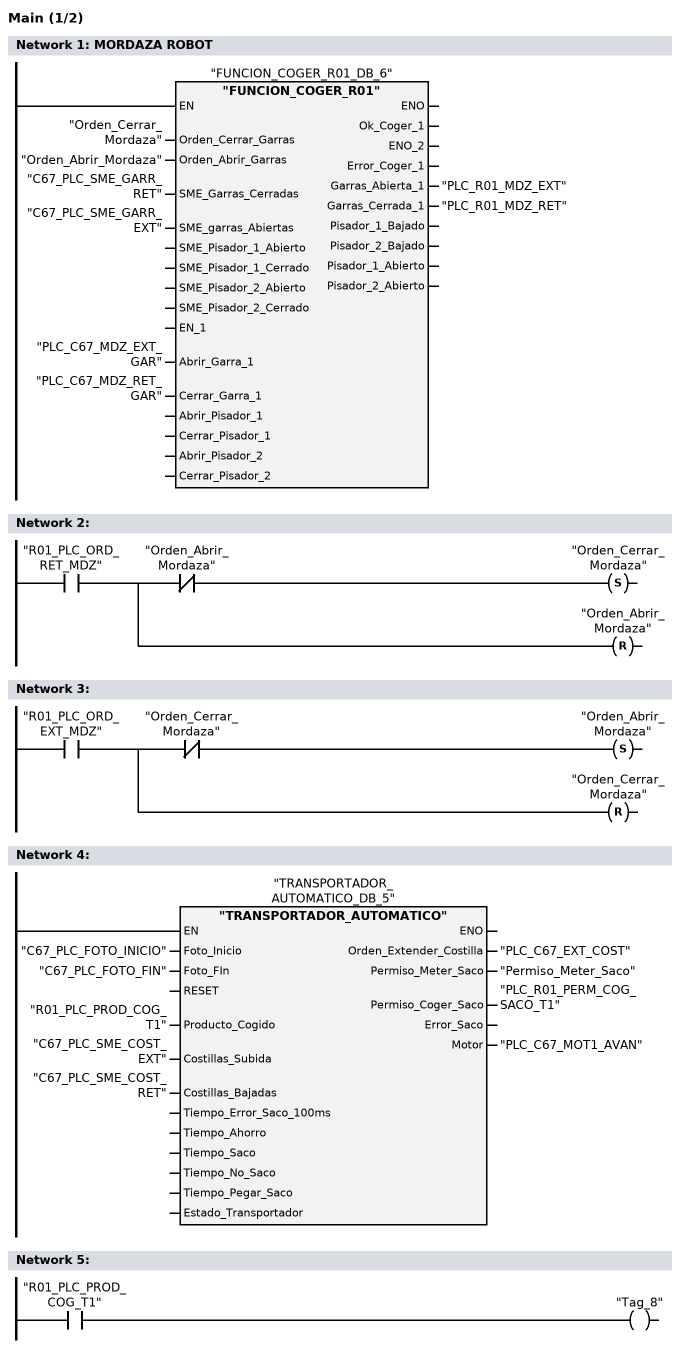
   RUNG wire#powerrail
      "FUNCION_COGER_R01_DB_6"(Orden_Cerrar_Garras := "Orden_Cerrar_Mordaza", Orden_Abrir_Garras := "Orden_Abrir_Mordaza", SME_Garras_Cerradas := "C67_PLC_SME_GARR_RET", SME_garras_Abiertas := "C67_PLC_SME_GARR_EXT", SME_Pisador_1_Abierto :=, SME_Pisador_1_Cerrado :=, SME_Pisador_2_Abierto :=, SME_Pisador_2_Cerrado :=, EN_1 :=, Abrir_Garra_1 := "PLC_C67_MDZ_EXT_GAR", Cerrar_Garra_1 := "PLC_C67_MDZ_RET_GAR", Abrir_Pisador_1 :=, Cerrar_Pisador_1 :=, Abrir_Pisador_2 :=, Cerrar_Pisador_2 :=, Ok_Coger_1 =>, ENO_2 =>, Error_Coger_1 =>, Garras_Abierta_1 => "PLC_R01_MDZ_EXT", Garras_Cerrada_1 => "PLC_R01_MDZ_RET", Pisador_1_Bajado =>, Pisador_2_Bajado =>, Pisador_1_Abierto =>, Pisador_2_Abierto =>)
   END_RUNG
   // the same network as SCL:
   "FUNCION_COGER_R01_DB_6"(Orden_Cerrar_Garras := "Orden_Cerrar_Mordaza",   // "FUNCION_COGER_R01"
                           Orden_Abrir_Garras := "Orden_Abrir_Mordaza",
                           SME_Garras_Cerradas := "C67_PLC_SME_GARR_RET",
                           SME_garras_Abiertas := "C67_PLC_SME_GARR_EXT",
                           Abrir_Garra_1 := "PLC_C67_MDZ_EXT_GAR",
                           Cerrar_Garra_1 := "PLC_C67_MDZ_RET_GAR",
                           Garras_Abierta_1 => "PLC_R01_MDZ_EXT",
                           Garras_Cerrada_1 => "PLC_R01_MDZ_RET");
END_REGION

REGION Network 2
   RUNG wire#powerrail
      Contact( "R01_PLC_ORD_RET_MDZ" )
      wire#w1
      I_Contact( "Orden_Abrir_Mordaza" )
      S_Coil( "Orden_Cerrar_Mordaza" )
   END_RUNG
   RUNG wire#w1
      R_Coil( "Orden_Abrir_Mordaza" )
   END_RUNG
   // the same network as SCL:
   IF "R01_PLC_ORD_RET_MDZ" AND NOT "Orden_Abrir_Mordaza" THEN "Orden_Cerrar_Mordaza" := TRUE; END_IF;
   IF "R01_PLC_ORD_RET_MDZ" THEN "Orden_Abrir_Mordaza" := FALSE; END_IF;
END_REGION

REGION Network 3
   RUNG wire#powerrail
      Contact( "R01_PLC_ORD_EXT_MDZ" )
      wire#w1
      I_Contact( "Orden_Cerrar_Mordaza" )
      S_Coil( "Orden_Abrir_Mordaza" )
   END_RUNG
   RUNG wire#w1
      R_Coil( "Orden_Cerrar_Mordaza" )
   END_RUNG
   // the same network as SCL:
   IF "R01_PLC_ORD_EXT_MDZ" AND NOT "Orden_Cerrar_Mordaza" THEN "Orden_Abrir_Mordaza" := TRUE; END_IF;
   IF "R01_PLC_ORD_EXT_MDZ" THEN "Orden_Cerrar_Mordaza" := FALSE; END_IF;
END_REGION

REGION Network 4
   RUNG wire#powerrail
      "TRANSPORTADOR_AUTOMATICO_DB_5"(Foto_Inicio := "C67_PLC_FOTO_INICIO", Foto_FIn := "C67_PLC_FOTO_FIN", RESET :=, Producto_Cogido := "R01_PLC_PROD_COG_T1", Costillas_Subida := "C67_PLC_SME_COST_EXT", Costillas_Bajadas := "C67_PLC_SME_COST_RET", Tiempo_Error_Saco_100ms :=, Tiempo_Ahorro :=, Tiempo_Saco :=, Tiempo_No_Saco :=, Tiempo_Pegar_Saco :=, Estado_Transportador :=, Orden_Extender_Costilla => "PLC_C67_EXT_COST", Permiso_Meter_Saco => "Permiso_Meter_Saco", Permiso_Coger_Saco => "PLC_R01_PERM_COG_SACO_T1", Error_Saco =>, Motor => "PLC_C67_MOT1_AVAN")
   END_RUNG
   // the same network as SCL:
   "TRANSPORTADOR_AUTOMATICO_DB_5"(Foto_Inicio := "C67_PLC_FOTO_INICIO",   // "TRANSPORTADOR_AUTOMATICO"
                           Foto_FIn := "C67_PLC_FOTO_FIN",
                           Producto_Cogido := "R01_PLC_PROD_COG_T1",
                           Costillas_Subida := "C67_PLC_SME_COST_EXT",
                           Costillas_Bajadas := "C67_PLC_SME_COST_RET",
                           Orden_Extender_Costilla => "PLC_C67_EXT_COST",
                           Permiso_Meter_Saco => "Permiso_Meter_Saco",
                           Permiso_Coger_Saco => "PLC_R01_PERM_COG_SACO_T1",
                           Motor => "PLC_C67_MOT1_AVAN");
END_REGION

REGION Network 5
   RUNG wire#powerrail
      Contact( "R01_PLC_PROD_COG_T1" )
      Coil( "Tag_8" )
   END_RUNG
   // the same network as SCL:
   "Tag_8" := "R01_PLC_PROD_COG_T1";
END_REGION

REGION Network 6
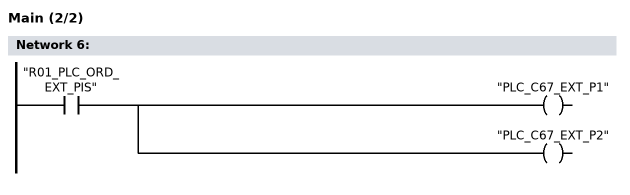
   RUNG wire#powerrail
      Contact( "R01_PLC_ORD_EXT_PIS" )
      wire#w1
      Coil( "PLC_C67_EXT_P1" )
   END_RUNG
   RUNG wire#w1
      Coil( "PLC_C67_EXT_P2" )
   END_RUNG
   // the same network as SCL:
   "PLC_C67_EXT_P1" := "R01_PLC_ORD_EXT_PIS";
   "PLC_C67_EXT_P2" := "R01_PLC_ORD_EXT_PIS";
END_REGION
END_ORGANIZATION_BLOCK